(* PLC project Cell Example , CTH FIX1 1.0, author CTH SS2 *)
(* stored: companyURL www.chalmers.se, creationDateTime 2008-03-19T20:31:26, version 1.0, modificationDateTime 2008-09-18T15:59:40, organization SS2, language en-US *)

TYPE BinaryPositions : ();
END_TYPE

TYPE HMIInput : ARRAY[0..0, 1..12] OF BOOL;
END_TYPE

FUNCTION ADD_E : INT
  VAR_INPUT
    Enable : BOOL := FALSE;
    IN1 : INT := 0;
    IN2 : INT := 0;
  END_VAR
  VAR_OUTPUT
    EnableO : BOOL := FALSE;
  END_VAR

(* LD diagram, written out as Structured Text *)
END_FUNCTION

FUNCTION DEC_E : INT
  VAR_INPUT
    Enable : BOOL;
  END_VAR
  VAR_OUTPUT
    EnableO : BOOL;
  END_VAR

(* LD diagram, written out as Structured Text *)
END_FUNCTION

FUNCTION MOVE_E : STRING
  VAR_INPUT
    Enable : BOOL := FALSE;
    IN : STRING;
  END_VAR
  VAR_OUTPUT
    EnableO : BOOL := FALSE;
  END_VAR

(* LD diagram, written out as Structured Text *)
END_FUNCTION

FUNCTION_BLOCK test4
  VAR_INPUT
    i1 : BOOL := FALSE;
  END_VAR
  VAR_OUTPUT
    o1 : BOOL := TRUE;
  END_VAR

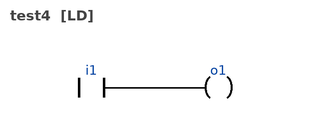
(* LD diagram, written out as Structured Text *)
o1 := i1;
END_FUNCTION_BLOCK

FUNCTION_BLOCK test2
  VAR_INPUT
    i : BOOL;
  END_VAR
  VAR_OUTPUT
    o : BOOL;
  END_VAR
  VAR
    internal1 : test4;
  END_VAR

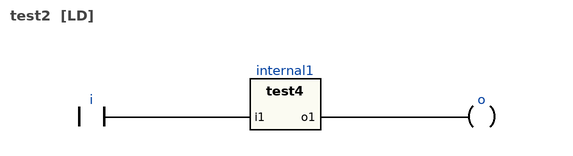
(* LD diagram, written out as Structured Text *)
internal1(i1 := i);
o := internal1.o1;
END_FUNCTION_BLOCK

FUNCTION_BLOCK test5
  VAR_INPUT
    in : BOOL;
  END_VAR
  VAR_OUTPUT
    ut : BOOL;
  END_VAR

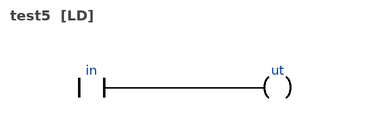
(* LD diagram, written out as Structured Text *)
ut := in;
END_FUNCTION_BLOCK

FUNCTION_BLOCK test3
  VAR_INPUT
    in1 : BOOL;
  END_VAR
  VAR_OUTPUT
    ut1 : BOOL;
  END_VAR
  VAR
    internal1 : test4;
    internal2 : test5;
  END_VAR

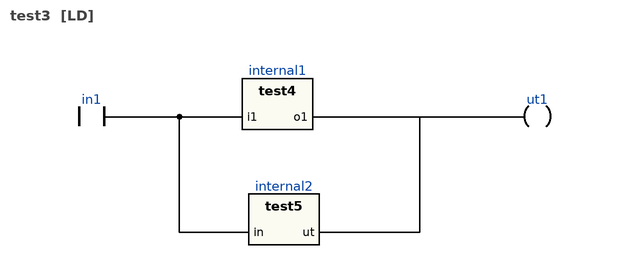
(* LD diagram, written out as Structured Text *)
internal1(i1 := in1);
internal2(in := in1);
ut1 := internal1.o1 OR internal2.ut;
END_FUNCTION_BLOCK

FUNCTION_BLOCK TestFB
  VAR_INPUT
    IN1 : BOOL := FALSE;
    IN2 : INT := 0;
    IN3 : BOOL := FALSE;
  END_VAR
  VAR_OUTPUT
    OUT1 : BOOL := FALSE;
    OUT2 : BOOL := FALSE;
    OUT3 : BOOL := FALSE;
    OUT4 : INT := 0;
  END_VAR
  VAR
    internal1 : test2;
    internal2 : test3;
  END_VAR

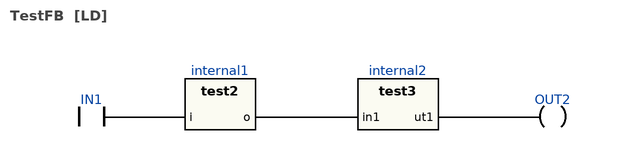
(* LD diagram, written out as Structured Text *)
internal1(i := IN1);
internal2(in1 := internal1.o);
OUT2 := internal2.ut1;
END_FUNCTION_BLOCK

FUNCTION_BLOCK RAC
  VAR_INPUT
    IN1 : BOOL := FALSE;
  END_VAR
  VAR_OUTPUT
    OUT : BOOL := FALSE;
  END_VAR
  VAR_INPUT
    IN2 : BOOL := TRUE;
  END_VAR
  VAR
    Var3 : BOOL := TRUE;
    IN4 : INT := 5;
  END_VAR
  VAR_OUTPUT
    State : STRING := 'Undefined';
  END_VAR
  VAR
    timer : TON;
    passedTime : TIME := 20;
    test : TestFB;
  END_VAR
  VAR_OUTPUT
    OUT2 : BOOL := TRUE;
  END_VAR
  VAR  (* added by the conversion: wires and edge detectors of the diagram *)
    _ADD_E24_ : ANY;
    _ADD_E24_OUT : INT;
    _MOVE_E26_ : ANY;
    _MOVE_E26_OUT : STRING;
    _DEC_E34_ : ANY;
    _DEC_E34_OUT : INT;
  END_VAR

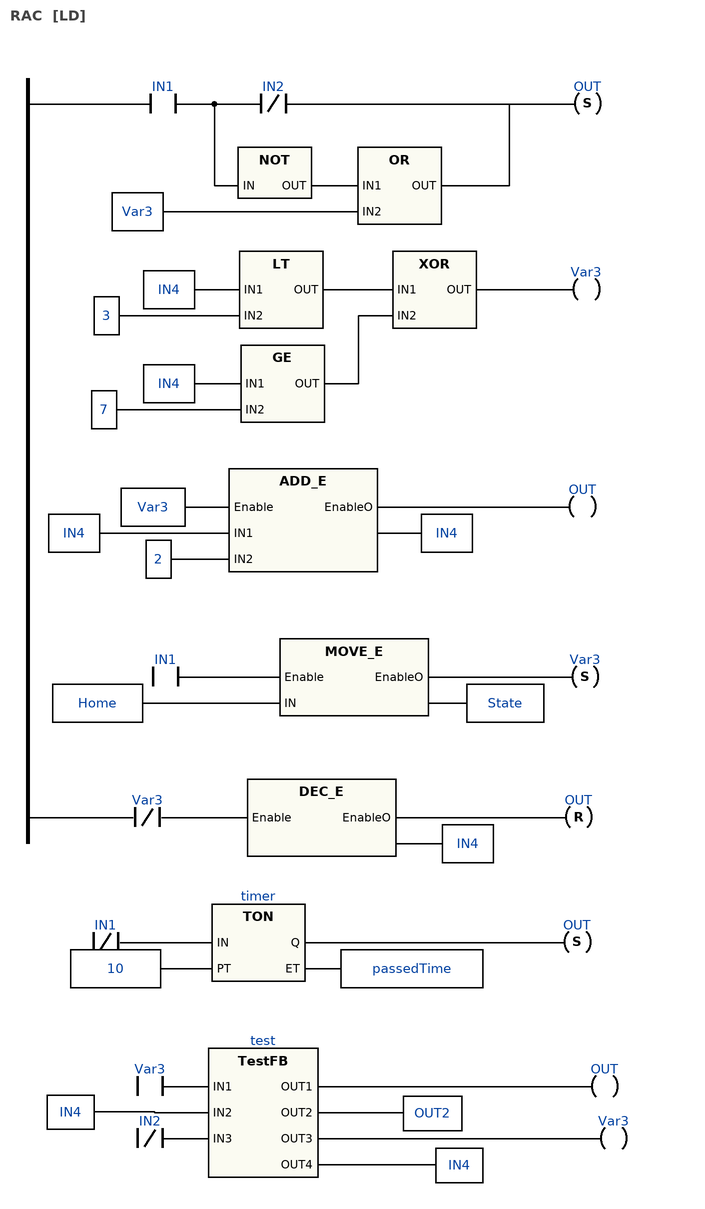
(* LD diagram, written out as Structured Text *)
IF IN1 AND NOT IN2 OR NOT IN1 OR Var3 THEN OUT := TRUE; END_IF;
Var3 := IN4 < 3 XOR IN4 >= 7;
_ADD_E24_OUT := ADD_E(Enable := Var3, IN1 := IN4, IN2 := 2,  => _ADD_E24_);
OUT := _ADD_E24_OUT;
IN4 := _ADD_E24_OUT;
_MOVE_E26_OUT := MOVE_E(Enable := IN1, IN := Home,  => _MOVE_E26_);
IF _MOVE_E26_OUT THEN Var3 := TRUE; END_IF;
State := _MOVE_E26_OUT;
_DEC_E34_OUT := DEC_E(Enable := NOT Var3,  => _DEC_E34_);
IF _DEC_E34_OUT THEN OUT := FALSE; END_IF;
IN4 := _DEC_E34_OUT;
timer(IN := NOT IN1, PT := 10);
IF timer.Q THEN OUT := TRUE; END_IF;
passedTime := timer.ET;
test(IN1 := Var3, IN2 := IN4, IN3 := NOT IN2);
OUT := test.OUT1;
OUT2 := test.OUT2;
Var3 := test.OUT3;
IN4 := test.OUT4;
END_FUNCTION_BLOCK

FUNCTION MOV_M : INT
  VAR_INPUT
    Enable : BOOL := FALSE;
    s_in : INT := 0;
  END_VAR
  VAR_OUTPUT
    EnableO : BOOL := FALSE;
  END_VAR

(* LD diagram, written out as Structured Text *)
END_FUNCTION

FUNCTION INCP_M : INT
  VAR_INPUT
    Enable : BOOL := FALSE;
  END_VAR
  VAR_OUTPUT
    EnableO : BOOL := FALSE;
  END_VAR

(* LD diagram, written out as Structured Text *)
END_FUNCTION

FUNCTION_BLOCK ESTOP
  VAR_INPUT
    ResetType : BOOL := FALSE;
    ChannelA : BOOL := TRUE;
    ChannelB : BOOL := TRUE;
    CircuitReset : BOOL := FALSE;
    FaultReset : BOOL := FALSE;
  END_VAR
  VAR_OUTPUT
    O1 : BOOL := FALSE;
    CI : BOOL := FALSE;
    CRHO : BOOL := FALSE;
    II : BOOL := FALSE;
    FP : BOOL := FALSE;
  END_VAR
  VAR
    RstOnlyByA : BOOL := FALSE;
    RstOnlyByB : BOOL := FALSE;
    RisingEdge1 : R_TRIG;
    RisingEdge2 : R_TRIG;
    Timer2 : TON;
    Timer1 : TON;
    RisingEdge3 : R_TRIG;
  END_VAR

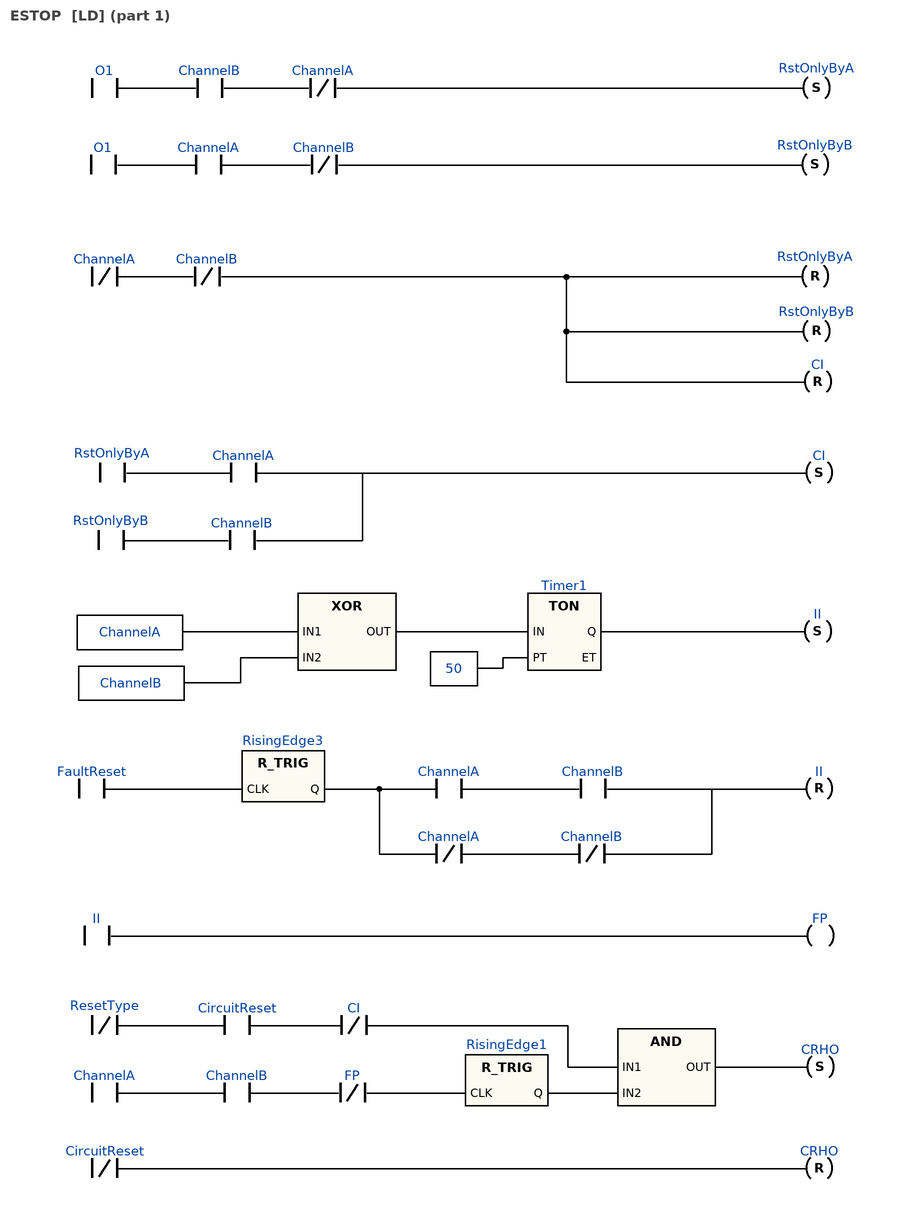
(* LD diagram, written out as Structured Text *)
IF O1 AND ChannelB AND NOT ChannelA THEN RstOnlyByA := TRUE; END_IF;
IF O1 AND ChannelA AND NOT ChannelB THEN RstOnlyByB := TRUE; END_IF;
IF NOT ChannelA AND NOT ChannelB THEN RstOnlyByA := FALSE; END_IF;
IF NOT ChannelA AND NOT ChannelB THEN RstOnlyByB := FALSE; END_IF;
IF NOT ChannelA AND NOT ChannelB THEN CI := FALSE; END_IF;
IF RstOnlyByA AND ChannelA OR RstOnlyByB AND ChannelB THEN CI := TRUE; END_IF;
Timer1(IN := ChannelA XOR ChannelB, PT := 50);
IF Timer1.Q THEN II := TRUE; END_IF;
RisingEdge3(CLK := FaultReset);
IF RisingEdge3.Q AND (ChannelA AND ChannelB OR NOT ChannelA AND NOT ChannelB) THEN II := FALSE; END_IF;
FP := II;
RisingEdge1(CLK := ChannelA AND ChannelB AND NOT FP);
IF NOT ResetType AND CircuitReset AND NOT CI AND RisingEdge1.Q THEN CRHO := TRUE; END_IF;
IF NOT CircuitReset THEN CRHO := FALSE; END_IF;
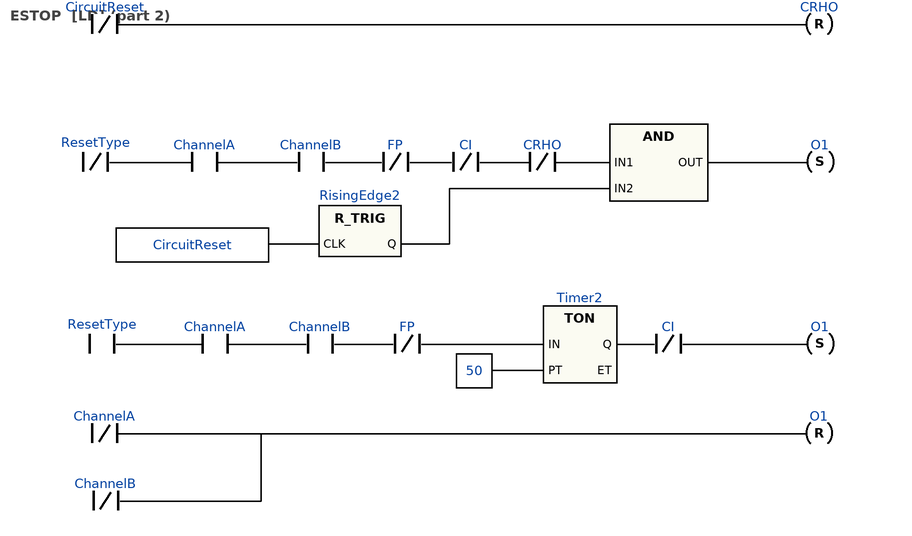
RisingEdge2(CLK := CircuitReset);
IF NOT ResetType AND ChannelA AND ChannelB AND NOT FP AND NOT CI AND NOT CRHO AND RisingEdge2.Q THEN O1 := TRUE; END_IF;
Timer2(IN := ResetType AND ChannelA AND ChannelB AND NOT FP, PT := 50);
IF Timer2.Q AND NOT CI THEN O1 := TRUE; END_IF;
IF NOT ChannelA OR NOT ChannelB THEN O1 := FALSE; END_IF;
END_FUNCTION_BLOCK

FUNCTION_BLOCK ENPEN
  VAR_INPUT
    ResetType : BOOL := FALSE;
    ChannelA : BOOL := TRUE;
    ChannelB : BOOL := TRUE;
    CircuitReset : BOOL := FALSE;
    FaultReset : BOOL := FALSE;
  END_VAR
  VAR_OUTPUT
    O1 : BOOL := FALSE;
    CI : BOOL := FALSE;
    CRHO : BOOL := FALSE;
    II : BOOL := FALSE;
    FP : BOOL := FALSE;
  END_VAR
  VAR
    RstOnlyByA : BOOL := FALSE;
    RstOnlyByB : BOOL := FALSE;
    CircuitReset_pre : BOOL := FALSE;
    RisingEdge1 : R_TRIG;
    RisingEdge2 : R_TRIG;
    Timer2 : TON;
    Timer1 : TON;
  END_VAR

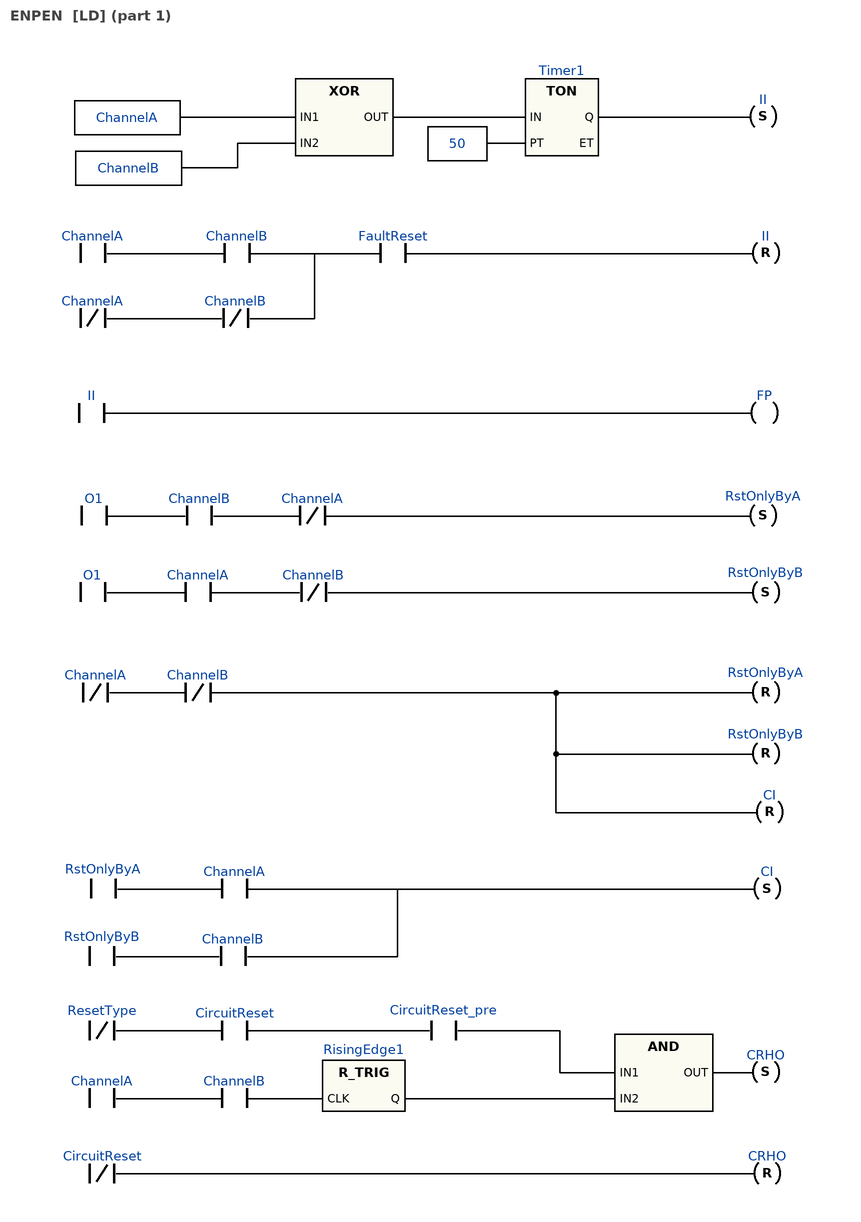
(* LD diagram, written out as Structured Text *)
Timer1(IN := ChannelA XOR ChannelB, PT := 50);
IF Timer1.Q THEN II := TRUE; END_IF;
IF (ChannelA AND ChannelB OR NOT ChannelA AND NOT ChannelB) AND FaultReset THEN II := FALSE; END_IF;
FP := II;
IF O1 AND ChannelB AND NOT ChannelA THEN RstOnlyByA := TRUE; END_IF;
IF O1 AND ChannelA AND NOT ChannelB THEN RstOnlyByB := TRUE; END_IF;
IF NOT ChannelA AND NOT ChannelB THEN RstOnlyByA := FALSE; END_IF;
IF NOT ChannelA AND NOT ChannelB THEN RstOnlyByB := FALSE; END_IF;
IF NOT ChannelA AND NOT ChannelB THEN CI := FALSE; END_IF;
IF RstOnlyByA AND ChannelA OR RstOnlyByB AND ChannelB THEN CI := TRUE; END_IF;
RisingEdge1(CLK := ChannelA AND ChannelB);
IF NOT ResetType AND CircuitReset AND CircuitReset_pre AND RisingEdge1.Q THEN CRHO := TRUE; END_IF;
IF NOT CircuitReset THEN CRHO := FALSE; END_IF;
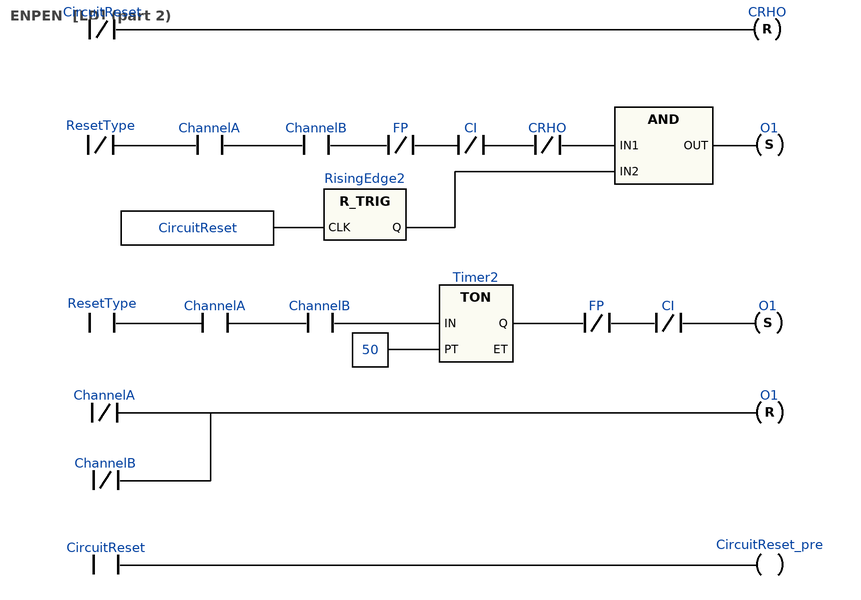
RisingEdge2(CLK := CircuitReset);
IF NOT ResetType AND ChannelA AND ChannelB AND NOT FP AND NOT CI AND NOT CRHO AND RisingEdge2.Q THEN O1 := TRUE; END_IF;
Timer2(IN := ResetType AND ChannelA AND ChannelB, PT := 50);
IF Timer2.Q AND NOT FP AND NOT CI THEN O1 := TRUE; END_IF;
IF NOT ChannelA OR NOT ChannelB THEN O1 := FALSE; END_IF;
CircuitReset_pre := CircuitReset;
END_FUNCTION_BLOCK

FUNCTION_BLOCK FPMS
  VAR
    NMCondition : BOOL := FALSE;
    MMSCondition : BOOL := FALSE;
  END_VAR
  VAR_INPUT
    FaultReset : BOOL := FALSE;
  END_VAR
  VAR_OUTPUT
    NM : BOOL := FALSE;
    FP : BOOL := FALSE;
  END_VAR
  VAR
    Timer1 : TON;
  END_VAR
  VAR_INPUT
    Input1 : BOOL := FALSE;
    Input2 : BOOL := FALSE;
    Input3 : BOOL := FALSE;
    Input4 : BOOL := FALSE;
    Input5 : BOOL := FALSE;
  END_VAR
  VAR_OUTPUT
    MMS : BOOL := FALSE;
  END_VAR
  VAR
    Timer2 : TON;
  END_VAR
  VAR_OUTPUT
    O1 : BOOL := FALSE;
    O2 : BOOL := FALSE;
    O3 : BOOL := FALSE;
    O4 : BOOL := FALSE;
    O5 : BOOL := FALSE;
  END_VAR
  VAR
    RisingEdge1 : R_TRIG;
    RisingEdge2 : R_TRIG;
  END_VAR

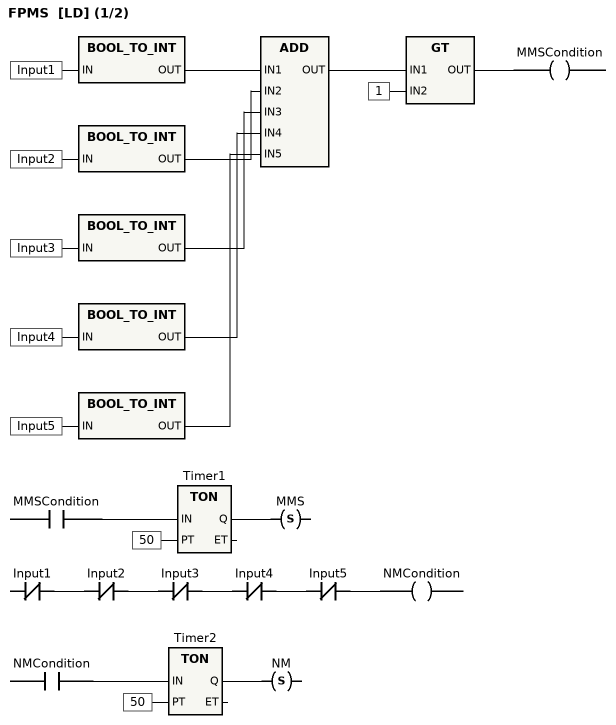
(* LD diagram, written out as Structured Text *)
MMSCondition := BOOL_TO_INT(Input1) + BOOL_TO_INT(Input2) + BOOL_TO_INT(Input3) + BOOL_TO_INT(Input4) + BOOL_TO_INT(Input5) > 1;
NMCondition := NOT Input1 AND NOT Input2 AND NOT Input3 AND NOT Input4 AND NOT Input5;
Timer1(IN := MMSCondition, PT := 50);
IF Timer1.Q THEN MMS := TRUE; END_IF;
Timer2(IN := NMCondition, PT := 50);
IF Timer2.Q THEN NM := TRUE; END_IF;
RisingEdge1(CLK := FaultReset);
IF RisingEdge1.Q AND NOT NMCondition THEN NM := FALSE; END_IF;
RisingEdge2(CLK := FaultReset);
IF RisingEdge2.Q AND NOT MMSCondition THEN MMS := FALSE; END_IF;
FP := NM OR MMS;
O1 := Input1 AND NOT Input2 AND NOT Input3 AND NOT Input4 AND NOT Input5 OR (NMCondition OR MMSCondition) AND O1;
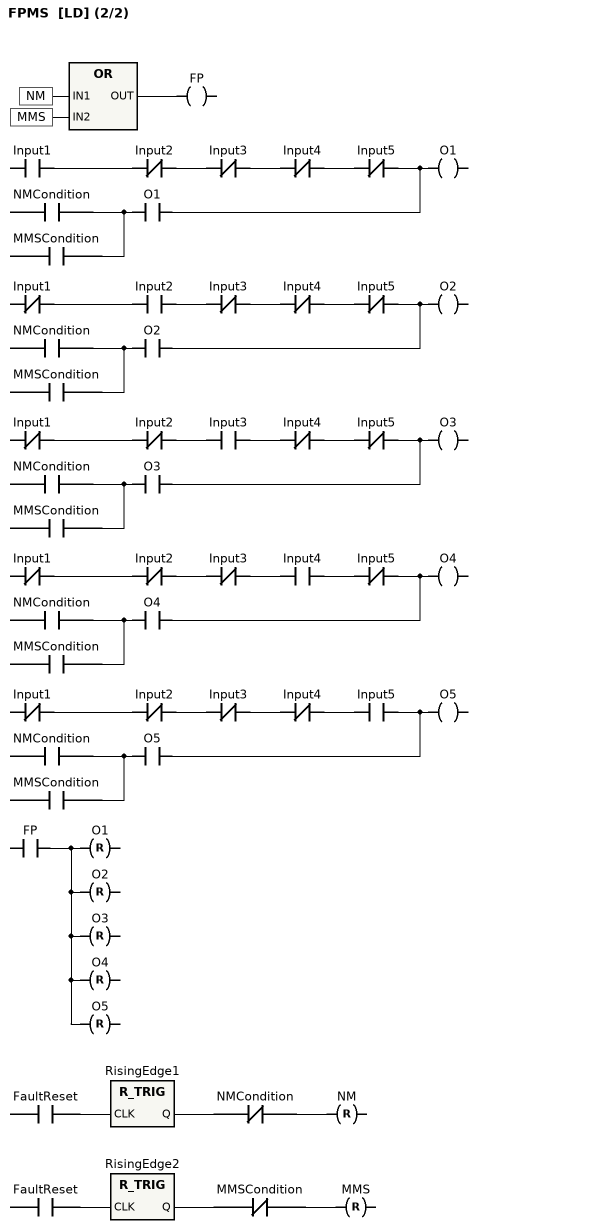
O2 := NOT Input1 AND Input2 AND NOT Input3 AND NOT Input4 AND NOT Input5 OR (NMCondition OR MMSCondition) AND O2;
O3 := NOT Input1 AND NOT Input2 AND Input3 AND NOT Input4 AND NOT Input5 OR (NMCondition OR MMSCondition) AND O3;
O4 := NOT Input1 AND NOT Input2 AND NOT Input3 AND Input4 AND NOT Input5 OR (NMCondition OR MMSCondition) AND O4;
O5 := NOT Input1 AND NOT Input2 AND NOT Input3 AND NOT Input4 AND Input5 OR (NMCondition OR MMSCondition) AND O5;
IF FP THEN O1 := FALSE; END_IF;
IF FP THEN O2 := FALSE; END_IF;
IF FP THEN O3 := FALSE; END_IF;
IF FP THEN O4 := FALSE; END_IF;
IF FP THEN O5 := FALSE; END_IF;
END_FUNCTION_BLOCK

FUNCTION_BLOCK RIN
  VAR_INPUT
    ResetType : BOOL := FALSE;
    ChannelA : BOOL := TRUE;
    ChannelB : BOOL := TRUE;
    CircuitReset : BOOL := FALSE;
    FaultReset : BOOL := FALSE;
  END_VAR
  VAR_OUTPUT
    O1 : BOOL := FALSE;
    CI : BOOL := FALSE;
    CRHO : BOOL := FALSE;
    II : BOOL := FALSE;
    FP : BOOL := FALSE;
  END_VAR
  VAR
    RstOnlyByA : BOOL := FALSE;
    RstOnlyByB : BOOL := FALSE;
    CircuitReset_pre : BOOL := FALSE;
    RisingEdge1 : R_TRIG;
    RisingEdge2 : R_TRIG;
    Timer2 : TON;
    Timer1 : TON;
  END_VAR
  VAR_TEMP
    Spec_SettingO1 : BOOL;
    Spec_ResettingO1 : BOOL;
    Spec_NotSettingO1 : BOOL;
    O1_previous : BOOL;
  END_VAR

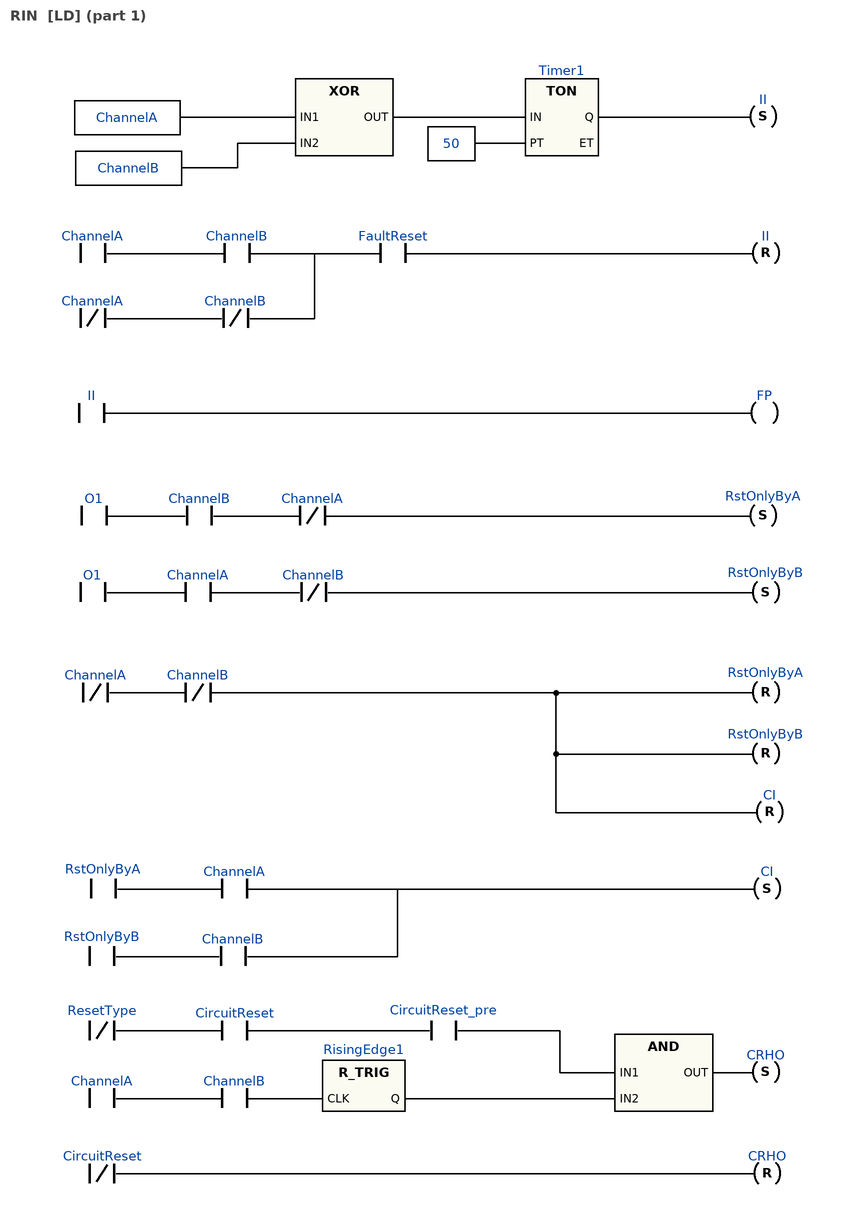
(* LD diagram, written out as Structured Text *)
Timer1(IN := ChannelA XOR ChannelB, PT := 50);
IF Timer1.Q THEN II := TRUE; END_IF;
IF (ChannelA AND ChannelB OR NOT ChannelA AND NOT ChannelB) AND FaultReset THEN II := FALSE; END_IF;
FP := II;
IF O1 AND ChannelB AND NOT ChannelA THEN RstOnlyByA := TRUE; END_IF;
IF O1 AND ChannelA AND NOT ChannelB THEN RstOnlyByB := TRUE; END_IF;
IF NOT ChannelA AND NOT ChannelB THEN RstOnlyByA := FALSE; END_IF;
IF NOT ChannelA AND NOT ChannelB THEN RstOnlyByB := FALSE; END_IF;
IF NOT ChannelA AND NOT ChannelB THEN CI := FALSE; END_IF;
IF RstOnlyByA AND ChannelA OR RstOnlyByB AND ChannelB THEN CI := TRUE; END_IF;
RisingEdge1(CLK := ChannelA AND ChannelB);
IF NOT ResetType AND CircuitReset AND CircuitReset_pre AND RisingEdge1.Q THEN CRHO := TRUE; END_IF;
IF NOT CircuitReset THEN CRHO := FALSE; END_IF;
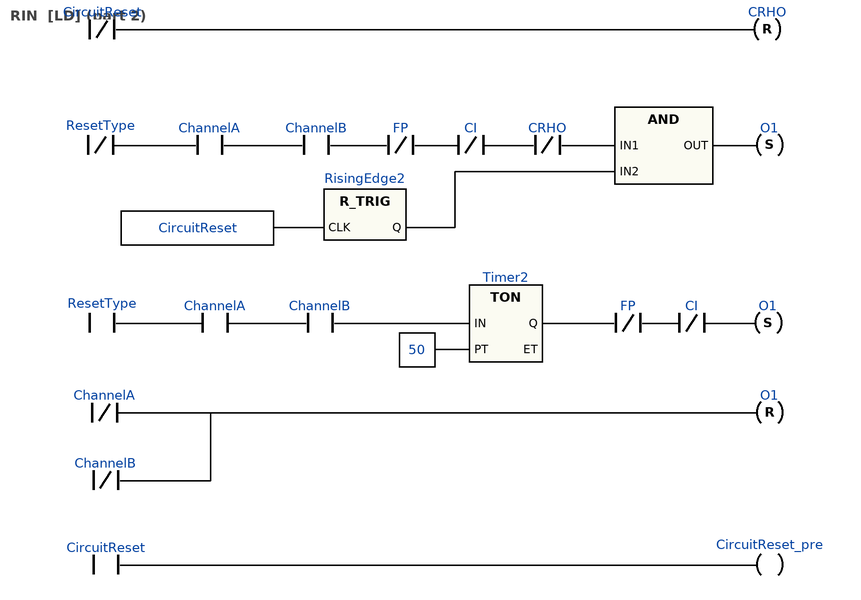
RisingEdge2(CLK := CircuitReset);
IF NOT ResetType AND ChannelA AND ChannelB AND NOT FP AND NOT CI AND NOT CRHO AND RisingEdge2.Q THEN O1 := TRUE; END_IF;
Timer2(IN := ResetType AND ChannelA AND ChannelB, PT := 50);
IF Timer2.Q AND NOT FP AND NOT CI THEN O1 := TRUE; END_IF;
IF NOT ChannelA OR NOT ChannelB THEN O1 := FALSE; END_IF;
CircuitReset_pre := CircuitReset;
END_FUNCTION_BLOCK

FUNCTION Always : BOOL
  VAR_INPUT
     : BOOL;
  END_VAR

(* LD diagram, written out as Structured Text *)
END_FUNCTION

FUNCTION Sometime : BOOL
  VAR_INPUT
     : BOOL;
  END_VAR

(* LD diagram, written out as Structured Text *)
END_FUNCTION

FUNCTION Never : BOOL
  VAR_INPUT
     : BOOL;
  END_VAR

(* LD diagram, written out as Structured Text *)
END_FUNCTION

FUNCTION Imply : BOOL
  VAR_INPUT
    IfTrue : BOOL;
    ThenTrue : BOOL;
  END_VAR

(* LD diagram, written out as Structured Text *)
END_FUNCTION

FUNCTION SteadyExpressionT : BOOL
  VAR_INPUT
    HeldTrueForXMilliSeconds : BOOL;
    X : INT := 10;
  END_VAR

(* LD diagram, written out as Structured Text *)
END_FUNCTION

FUNCTION SteadyExpressionSC : BOOL
  VAR_INPUT
    RemainTrueForXScanCycles : BOOL;
    X : INT := 1;
  END_VAR

(* LD diagram, written out as Structured Text *)
END_FUNCTION

FUNCTION_BLOCK Implies
  VAR_INPUT
    IfTrue : BOOL;
  END_VAR
  VAR_OUTPUT
    ThenTrue : BOOL;
  END_VAR

(* LD diagram, written out as Structured Text *)
END_FUNCTION_BLOCK

FUNCTION WhileNot : BOOL
  VAR_INPUT
    RemainTrue : BOOL;
    WhileNot : BOOL;
  END_VAR

(* LD diagram, written out as Structured Text *)
END_FUNCTION

FUNCTION MOV_E_Int : INT
  VAR_INPUT
    Enable : BOOL := FALSE;
    Source : INT := 0;
  END_VAR
  VAR_OUTPUT
    EnableO : BOOL := FALSE;
  END_VAR

(* LD diagram, written out as Structured Text *)
END_FUNCTION

FUNCTION_BLOCK TOF_RSLogix
  VAR_INPUT
    TimerOffDelay : BOOL;
    Preset : INT;
  END_VAR
  VAR_OUTPUT
    EnableO : BOOL := FALSE;
    DN : BOOL := FALSE;
    ACC : INT := 0;
    TT : BOOL := FALSE;
  END_VAR
  VAR
    TON1 : TON;
  END_VAR

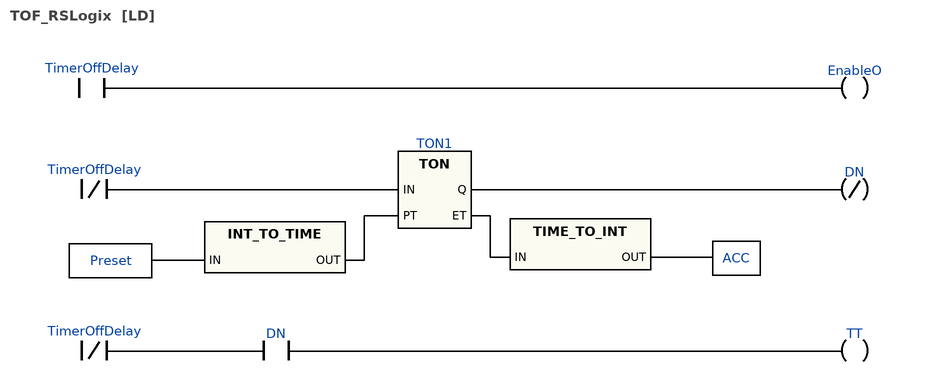
(* LD diagram, written out as Structured Text *)
EnableO := TimerOffDelay;
TON1(IN := NOT TimerOffDelay, PT := INT_TO_TIME(Preset));
DN := NOT TON1.Q;
ACC := TIME_TO_INT(TON1.ET);
TT := NOT TimerOffDelay AND DN;
END_FUNCTION_BLOCK

FUNCTION_BLOCK TON_RSLogix
  VAR_INPUT
    TimerOnDelay : BOOL := FALSE;
    Preset : INT := 0;
  END_VAR
  VAR_OUTPUT
    EnableO : BOOL := FALSE;
    DN : BOOL := FALSE;
    ACC : INT := 0;
    TT : BOOL := FALSE;
  END_VAR
  VAR
    TON1 : TON;
  END_VAR

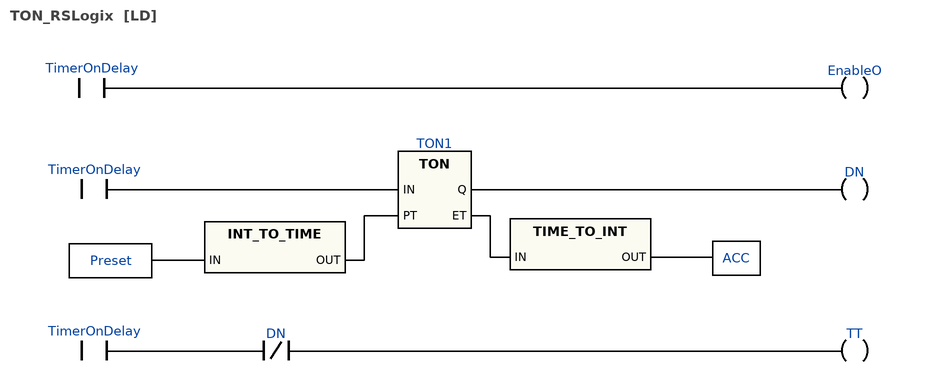
(* LD diagram, written out as Structured Text *)
EnableO := TimerOnDelay;
TON1(IN := TimerOnDelay, PT := INT_TO_TIME(Preset));
DN := TON1.Q;
ACC := TIME_TO_INT(TON1.ET);
TT := TimerOnDelay AND NOT DN;
END_FUNCTION_BLOCK

FUNCTION_BLOCK HMI_Safety
  VAR_IN_OUT
    ESTOP_FP : BOOL := FALSE;
    CommOK : BOOL := FALSE;
  END_VAR
  VAR_INPUT
    FirstScanOneShot : BOOL;
    NoEStopCHA : BOOL;
    NoEStopCHB : BOOL;
  END_VAR
  VAR_OUTPUT
    ESTOP_FaultReset : BOOL := FALSE;
    ESTOP_O1 : BOOL := FALSE;
    NoEstop : BOOL := FALSE;
  END_VAR
  VAR_INPUT
    AutoModeS : BOOL;
    ManModeS : BOOL;
  END_VAR
  VAR_IN_OUT
    AutoMan_FP : BOOL := FALSE;
  END_VAR
  VAR_OUTPUT
    AutoMan_FaultReset : BOOL := FALSE;
    AutoManDebounce_PRE : INT := 200;
    AutoManDebounce_TT : BOOL := FALSE;
  END_VAR
  VAR_IN_OUT
    Pos1Int : BOOL := FALSE;
    Pos2Int : BOOL := FALSE;
  END_VAR
  VAR_OUTPUT
    AutoMan_O1 : BOOL := FALSE;
    AutoMan_O2 : BOOL := FALSE;
    AutoMode : BOOL := FALSE;
    ManualMode : BOOL := FALSE;
  END_VAR
  VAR_IN_OUT
    PendantOK_FP : BOOL := FALSE;
  END_VAR
  VAR_OUTPUT
    PendantOK_FaultReset : BOOL := FALSE;
  END_VAR
  VAR_INPUT
    E130CREP : BOOL;
    E134CREP : BOOL;
    HMI_Select : BOOL;
  END_VAR
  VAR_IN_OUT
    Selected : BOOL := FALSE;
  END_VAR
  VAR_INPUT
    HMI_SelectionOK : BOOL;
    Gates_SelectAvail : BOOL;
    EnablePB : BOOL;
  END_VAR
  VAR_IN_OUT
    Enable : BOOL := FALSE;
    PHMIEnable : BOOL := FALSE;
    EnableAntiRepeat : BOOL := FALSE;
  END_VAR
  VAR_OUTPUT
    EnableTmr_PRE : INT := 600;
    EnableTmr_DN : BOOL := FALSE;
  END_VAR
  VAR_INPUT
    OneHMIEnabled : BOOL;
    Gates_OneRobotToolMinorReq : BOOL;
    OneHMIMode : BOOL;
  END_VAR
  VAR_OUTPUT
    PendEnable : BOOL := FALSE;
    PendOk : BOOL := FALSE;
  END_VAR
  VAR_INPUT
    AlwaysOff : BOOL;
    FltBcn : BOOL;
  END_VAR
  VAR_OUTPUT
    O_FaultLT : BOOL := FALSE;
  END_VAR
  VAR_INPUT
    ResetLT : BOOL;
  END_VAR
  VAR_OUTPUT
    O_ResetLT : BOOL := FALSE;
  END_VAR
  VAR_INPUT
    AutoInitLT : BOOL;
  END_VAR
  VAR_OUTPUT
    O_AutoInitLT : BOOL := FALSE;
  END_VAR
  VAR_INPUT
    CombinedStatus : BOOL;
  END_VAR
  VAR_OUTPUT
    NoSafetyFaults : BOOL := FALSE;
  END_VAR
  VAR_IN_OUT
    BackCheck_NoEStop : BOOL := FALSE;
    BackCheck_NoSafetyFaults : BOOL := FALSE;
  END_VAR
  VAR
    ESTOP1 : ESTOP;
    TOF1 : TOF_RSLogix;
    FPMS1 : FPMS;
    ENPEN1 : ENPEN;
    TON1 : TON_RSLogix;
  END_VAR
  VAR_OUTPUT
    ESTOP_CI : BOOL := FALSE;
    ESTOP_CRHO : BOOL := FALSE;
    ESTOP_II : BOOL := FALSE;
  END_VAR
  VAR  (* added by the conversion: wires and edge detectors of the diagram *)
    _MOV_E_Int30_ : ANY;
    _MOV_E_Int30_OUT : INT;
    _MOV_E_Int83_ : ANY;
    _MOV_E_Int83_OUT : INT;
  END_VAR

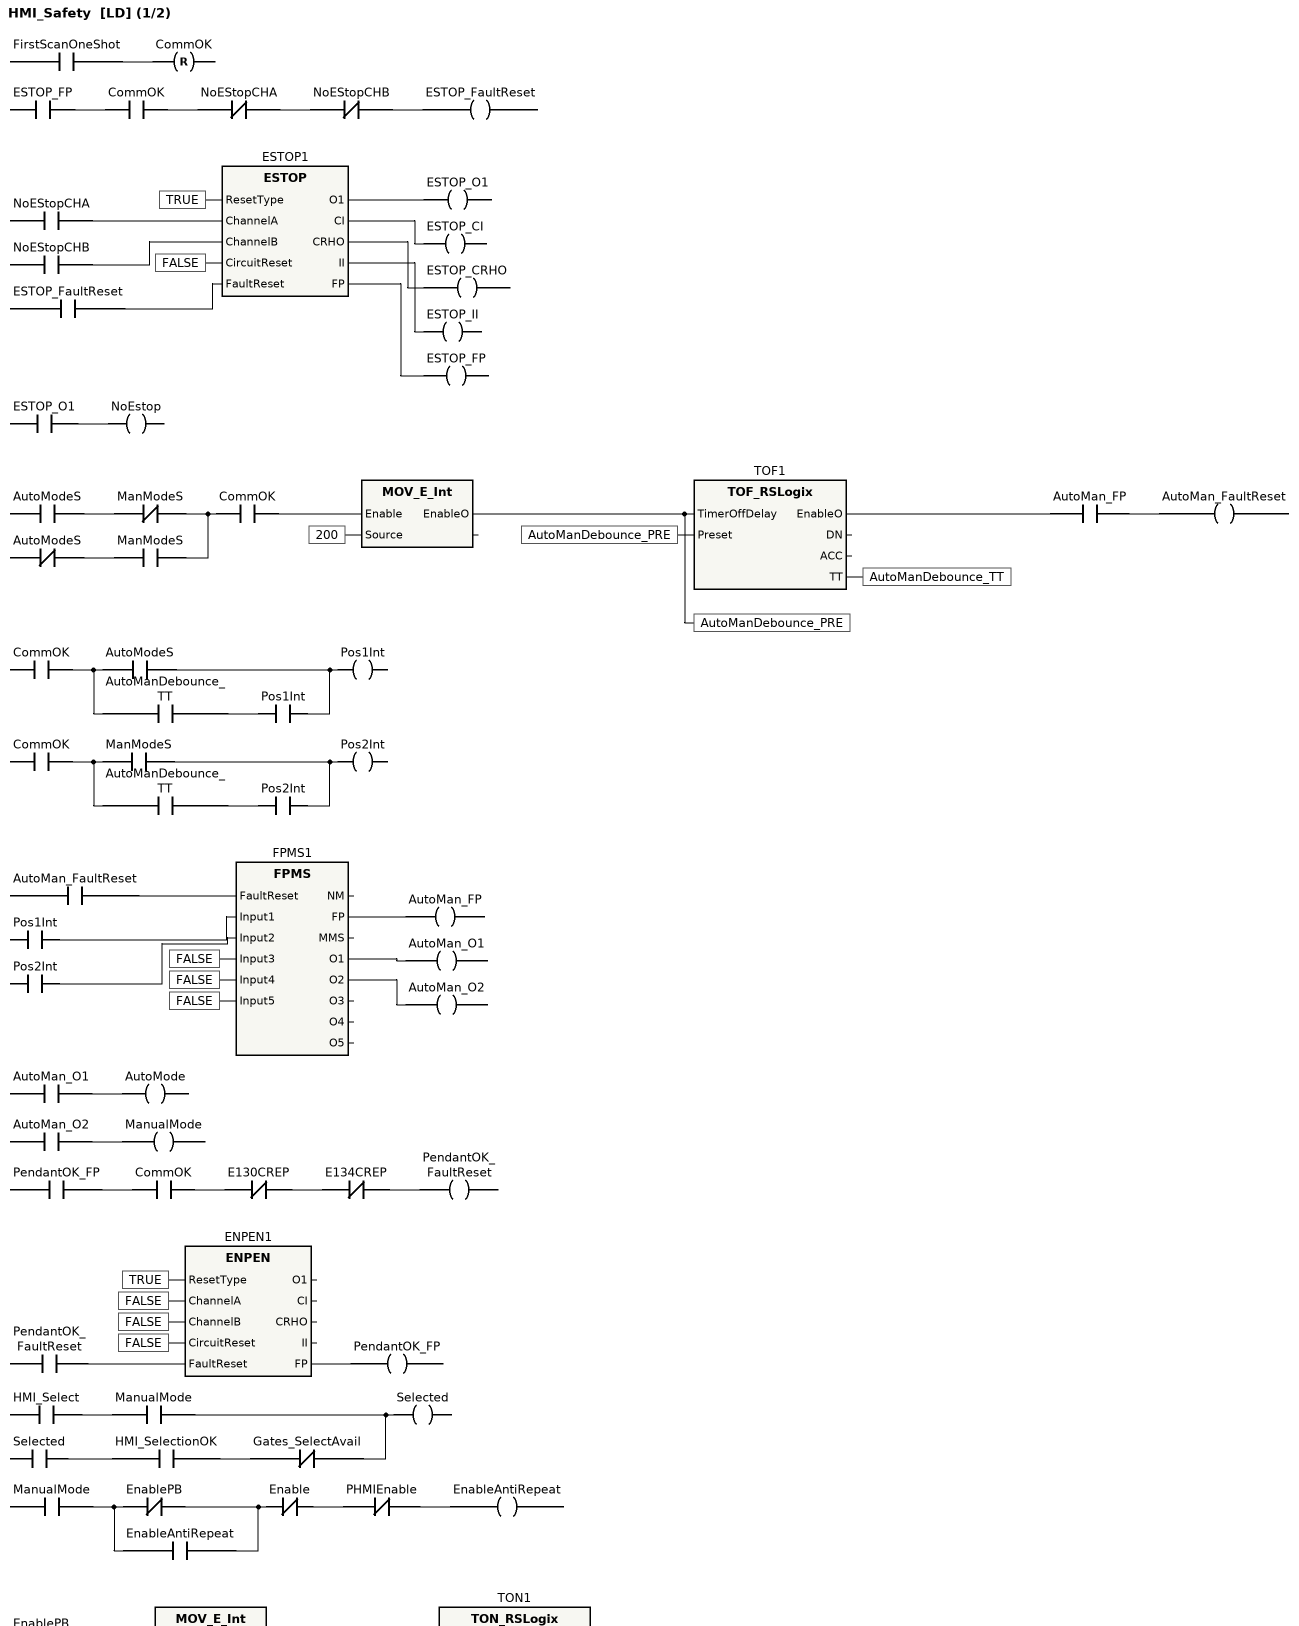
(* LD diagram, written out as Structured Text *)
IF FirstScanOneShot THEN CommOK := FALSE; END_IF;
ESTOP_FaultReset := ESTOP_FP AND CommOK AND NOT NoEStopCHA AND NOT NoEStopCHB;
ESTOP1(ResetType := TRUE, ChannelA := NoEStopCHA, ChannelB := NoEStopCHB, CircuitReset := FALSE, FaultReset := ESTOP_FaultReset);
ESTOP_O1 := ESTOP1.O1;
ESTOP_CI := ESTOP1.CI;
ESTOP_CRHO := ESTOP1.CRHO;
ESTOP_II := ESTOP1.II;
ESTOP_FP := ESTOP1.FP;
NoEstop := ESTOP_O1;
_MOV_E_Int30_OUT := MOV_E_Int(Enable := (AutoModeS AND NOT ManModeS OR NOT AutoModeS AND ManModeS) AND CommOK, Source := 200,  => _MOV_E_Int30_);
TOF1(TimerOffDelay := _MOV_E_Int30_OUT, Preset := AutoManDebounce_PRE);
AutoMan_FaultReset := TOF1.EnableO AND AutoMan_FP;
AutoManDebounce_PRE := _MOV_E_Int30_OUT;
AutoManDebounce_TT := TOF1.TT;
Pos1Int := CommOK AND (AutoModeS OR AutoManDebounce_TT AND Pos1Int);
Pos2Int := CommOK AND (ManModeS OR AutoManDebounce_TT AND Pos2Int);
FPMS1(FaultReset := AutoMan_FaultReset, Input1 := Pos1Int, Input2 := Pos2Int, Input3 := FALSE, Input4 := FALSE, Input5 := FALSE);
AutoMan_FP := FPMS1.FP;
AutoMan_O1 := FPMS1.O1;
AutoMan_O2 := FPMS1.O2;
AutoMode := AutoMan_O1;
ManualMode := AutoMan_O2;
PendantOK_FaultReset := PendantOK_FP AND CommOK AND NOT E130CREP AND NOT E134CREP;
ENPEN1(ResetType := TRUE, ChannelA := FALSE, ChannelB := FALSE, CircuitReset := FALSE, FaultReset := PendantOK_FaultReset);
PendantOK_FP := ENPEN1.FP;
Selected := HMI_Select AND ManualMode OR Selected AND HMI_SelectionOK AND NOT Gates_SelectAvail;
EnableAntiRepeat := ManualMode AND (NOT EnablePB OR EnableAntiRepeat) AND NOT Enable AND NOT PHMIEnable;
_MOV_E_Int83_OUT := MOV_E_Int(Enable := EnablePB, Source := 600,  => _MOV_E_Int83_);
EnableTmr_PRE := _MOV_E_Int83_OUT;
TON1(TimerOnDelay := _MOV_E_Int83_OUT, Preset := EnableTmr_PRE);
EnableTmr_DN := TON1.DN;
Enable := ManualMode AND NOT EnableTmr_DN AND (EnableAntiRepeat OR Enable) AND EnablePB AND ((NOT Gates_OneRobotToolMinorReq OR Selected AND HMI_SelectionOK) AND OneHMIEnabled OR (Selected AND HMI_SelectionOK OR NOT Gates_OneRobotToolMinorReq) AND NOT OneHMIMode);
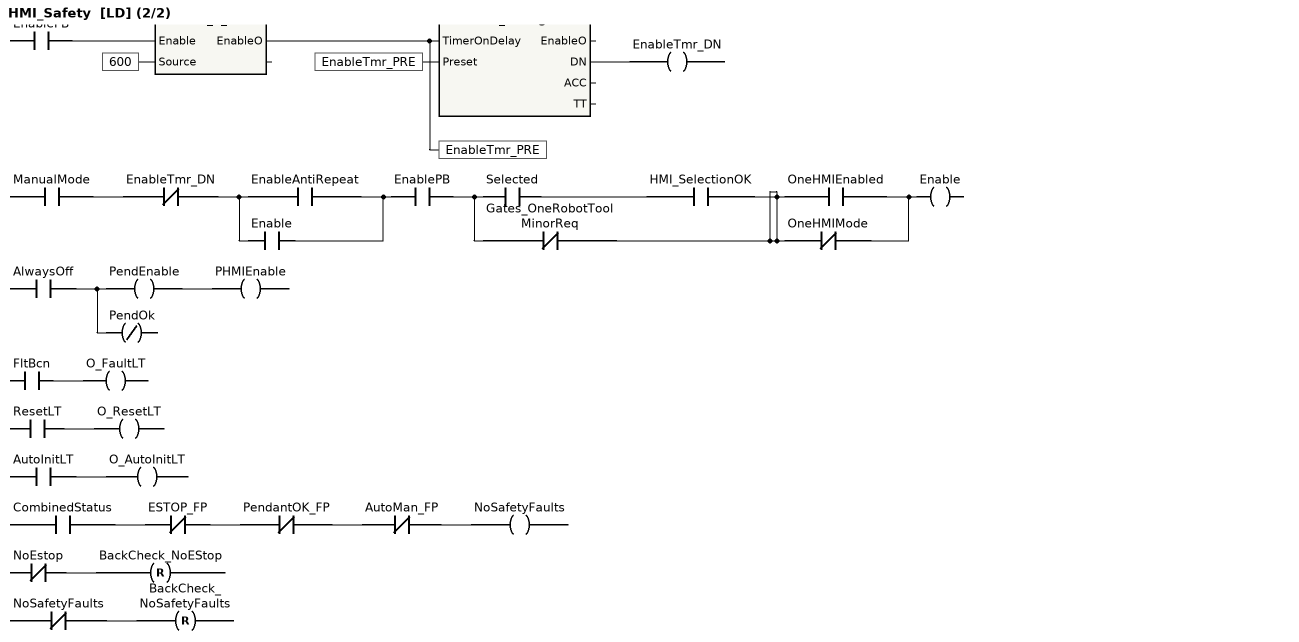
PendEnable := AlwaysOff;
PHMIEnable := AlwaysOff;
PendOk := NOT AlwaysOff;
O_FaultLT := FltBcn;
O_ResetLT := ResetLT;
O_AutoInitLT := AutoInitLT;
NoSafetyFaults := CombinedStatus AND NOT ESTOP_FP AND NOT PendantOK_FP AND NOT AutoMan_FP;
IF NOT NoEstop THEN BackCheck_NoEStop := FALSE; END_IF;
IF NOT NoSafetyFaults THEN BackCheck_NoSafetyFaults := FALSE; END_IF;
END_FUNCTION_BLOCK

FUNCTION_BLOCK PermGuard_Safety
  VAR_IN_OUT
    MuteSw12_FP : BOOL := FALSE;
    CommOK : BOOL := FALSE;
  END_VAR
  VAR_INPUT
    FirstScanOneShot : BOOL;
    SD1ClearChA : BOOL;
    SD1ClearChB : BOOL;
  END_VAR
  VAR_OUTPUT
    MuteSw12_FaultReset : BOOL := FALSE;
    MuteSw12_O1 : BOOL := FALSE;
  END_VAR
  VAR_INPUT
    AutoModeSS : BOOL;
    OverrideModeSS : BOOL;
  END_VAR
  VAR_IN_OUT
    AutoOverride_FP : BOOL := FALSE;
  END_VAR
  VAR_OUTPUT
    AutoOverride_FaultReset : BOOL := FALSE;
    AutoOverrideDebounce_PRE : INT := 50;
    AutoOverrideDebounce_TT : BOOL := FALSE;
  END_VAR
  VAR_IN_OUT
    Pos1Int : BOOL := FALSE;
    Pos2Int : BOOL := FALSE;
  END_VAR
  VAR_OUTPUT
    AutoOverride_O1 : BOOL := FALSE;
    AutoOverride_O2 : BOOL := FALSE;
  END_VAR
  VAR_IN_OUT
    GuardRst_FP : BOOL := FALSE;
  END_VAR
  VAR_OUTPUT
    GuardRst_FaultReset : BOOL := FALSE;
    OverrideLimit_PRE : INT := 50;
    OverrideLimit_DN : BOOL := FALSE;
  END_VAR
  VAR_INPUT
    CombinedStatus : BOOL;
  END_VAR
  VAR_OUTPUT
    NoSafetyFaults : BOOL := FALSE;
  END_VAR
  VAR_IN_OUT
    BackCheck_OneRobotEnable : BOOL := FALSE;
    BackCheck_NoSafetyFaults : BOOL := FALSE;
  END_VAR
  VAR
    MuteSw12 : ENPEN;
    AutoOverrideDebounce : TOF_RSLogix;
    AutoOverride : FPMS;
    GuardRst : RIN;
    OverrideLimit : TON_RSLogix;
  END_VAR
  VAR_OUTPUT
    MuteSw12_CI : BOOL := FALSE;
    MuteSw12_CRHO : BOOL := FALSE;
    MuteSw12_II : BOOL := FALSE;
  END_VAR
  VAR_INPUT
    P1 : BOOL;
    P2 : BOOL;
    P3 : BOOL;
    P4 : BOOL;
  END_VAR
  VAR_IN_OUT
    MuteSw34_FP : BOOL := FALSE;
  END_VAR
  VAR_OUTPUT
    MuteSw34_FaultReset : BOOL := FALSE;
    MuteSw34_O1 : BOOL := FALSE;
    MuteSw34_CI : BOOL := FALSE;
    MuteSw34_CRHO : BOOL := FALSE;
    MuteSw34_II : BOOL := FALSE;
  END_VAR
  VAR
    MuteSw34 : ENPEN;
  END_VAR
  VAR_INPUT
    MutingStatus : BOOL;
  END_VAR
  VAR_OUTPUT
    MuteSD : BOOL := FALSE;
    SDMuteLt : BOOL := FALSE;
  END_VAR
  VAR_INPUT
    LampTest : BOOL;
  END_VAR
  VAR_IN_OUT
    SD1_FP : BOOL := FALSE;
  END_VAR
  VAR_OUTPUT
    SD1_FaultReset : BOOL := FALSE;
    SD1_O1 : BOOL := FALSE;
    SD1_CI : BOOL := FALSE;
    SD1_CRHO : BOOL := FALSE;
    SD1_II : BOOL := FALSE;
  END_VAR
  VAR
    SD1 : RIN;
  END_VAR
  VAR_OUTPUT
    SD1Clear : BOOL := FALSE;
    AutoOverrideDebounce_DN : BOOL := FALSE;
    AutoOverrideDebounce_ACC : INT := 0;
    AutoOverride_NM : BOOL := FALSE;
    AutoOverride_MMS : BOOL := FALSE;
    ResetReady : BOOL := FALSE;
  END_VAR
  VAR_INPUT
    ResetGrdPB : BOOL;
  END_VAR
  VAR_OUTPUT
    GuardRst_O1 : BOOL := FALSE;
    GuardRst_CI : BOOL := FALSE;
    GuardRst_CRHO : BOOL := FALSE;
    GuardRst_II : BOOL := FALSE;
    GuardReset : BOOL := FALSE;
    ToolMinorEnable : BOOL := FALSE;
    NobotEnable : BOOL := FALSE;
    RobotServoEnable : BOOL := FALSE;
    OneRobotEnable : BOOL := FALSE;
    AutoOverrideDebounce_EN : BOOL := FALSE;
    OverrideLimit_EN : BOOL := FALSE;
    OverrideLimit_ACC : INT := 0;
    OverrideLimit_TT : BOOL := FALSE;
    ToolMajorEnable : BOOL := FALSE;
  END_VAR
  VAR_INPUT
    FlashNorm : BOOL;
  END_VAR
  VAR_OUTPUT
    GuardResetLt : BOOL := FALSE;
  END_VAR
  VAR_IN_OUT
    BackCheck_GateReset : BOOL := FALSE;
    BackCheck_ToolMinorEnable : BOOL := FALSE;
    BackCheck_ToolMajorEnable : BOOL := FALSE;
    BackCheck_NobotEnable : BOOL := FALSE;
    BackCheck_RobotServoEnable : BOOL := FALSE;
  END_VAR
  VAR  (* added by the conversion: wires and edge detectors of the diagram *)
    _MOV_E_Int30_ : ANY;
    _MOV_E_Int30_OUT : INT;
    _MOV_E_Int83_ : ANY;
    _MOV_E_Int83_OUT : INT;
  END_VAR

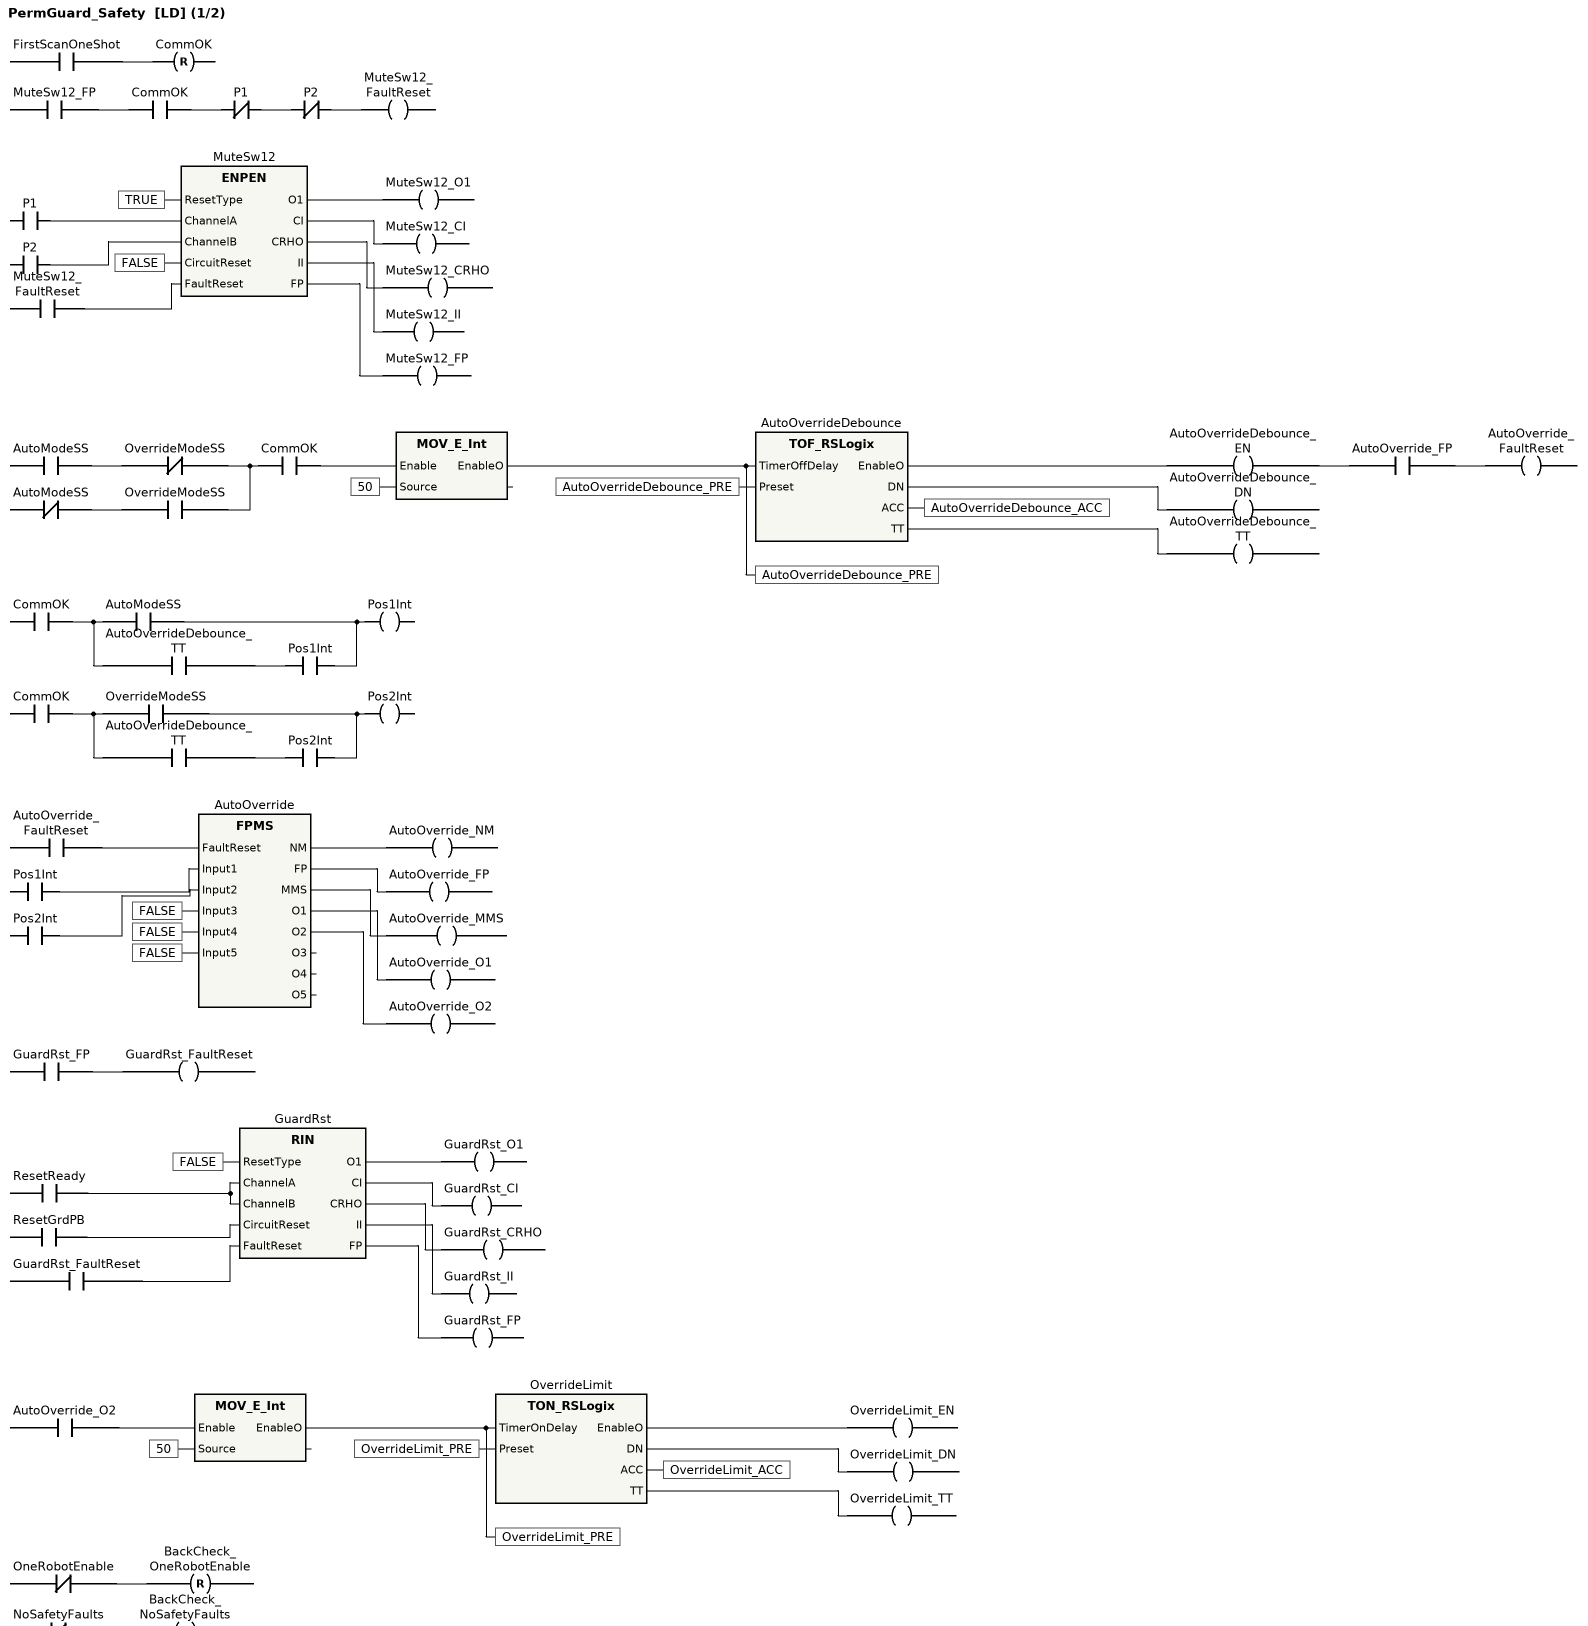
(* LD diagram, written out as Structured Text *)
IF FirstScanOneShot THEN CommOK := FALSE; END_IF;
MuteSw12_FaultReset := MuteSw12_FP AND CommOK AND NOT P1 AND NOT P2;
MuteSw12(ResetType := TRUE, ChannelA := P1, ChannelB := P2, CircuitReset := FALSE, FaultReset := MuteSw12_FaultReset);
MuteSw12_O1 := MuteSw12.O1;
MuteSw12_CI := MuteSw12.CI;
MuteSw12_CRHO := MuteSw12.CRHO;
MuteSw12_II := MuteSw12.II;
MuteSw12_FP := MuteSw12.FP;
MuteSw34_FaultReset := MuteSw34_FP AND CommOK AND NOT P3 AND NOT P4;
MuteSw34(ResetType := TRUE, ChannelA := P3, ChannelB := P4, CircuitReset := FALSE, FaultReset := MuteSw34_FaultReset);
MuteSw34_O1 := MuteSw34.O1;
MuteSw34_CI := MuteSw34.CI;
MuteSw34_CRHO := MuteSw34.CRHO;
MuteSw34_II := MuteSw34.II;
MuteSw34_FP := MuteSw34.FP;
MuteSD := (MuteSw12_O1 OR MuteSw34_O1) AND MutingStatus;
SDMuteLt := MuteSD OR LampTest;
SD1_FaultReset := SD1_FP AND CommOK AND NOT SD1ClearChA AND NOT SD1ClearChB;
SD1(ResetType := TRUE, ChannelA := SD1ClearChA, ChannelB := SD1ClearChB, CircuitReset := FALSE, FaultReset := SD1_FaultReset);
SD1_O1 := SD1.O1;
SD1_CI := SD1.CI;
SD1_CRHO := SD1.CRHO;
SD1_II := SD1.II;
SD1_FP := SD1.FP;
SD1Clear := SD1_O1;
_MOV_E_Int30_OUT := MOV_E_Int(Enable := (AutoModeSS AND NOT OverrideModeSS OR NOT AutoModeSS AND OverrideModeSS) AND CommOK, Source := 50,  => _MOV_E_Int30_);
AutoOverrideDebounce(TimerOffDelay := _MOV_E_Int30_OUT, Preset := AutoOverrideDebounce_PRE);
AutoOverrideDebounce_EN := AutoOverrideDebounce.EnableO;
AutoOverride_FaultReset := AutoOverrideDebounce.EnableO AND AutoOverride_FP;
AutoOverrideDebounce_PRE := _MOV_E_Int30_OUT;
AutoOverrideDebounce_DN := AutoOverrideDebounce.DN;
AutoOverrideDebounce_ACC := AutoOverrideDebounce.ACC;
AutoOverrideDebounce_TT := AutoOverrideDebounce.TT;
Pos1Int := CommOK AND (AutoModeSS OR AutoOverrideDebounce_TT AND Pos1Int);
Pos2Int := CommOK AND (OverrideModeSS OR AutoOverrideDebounce_TT AND Pos2Int);
AutoOverride(FaultReset := AutoOverride_FaultReset, Input1 := Pos1Int, Input2 := Pos2Int, Input3 := FALSE, Input4 := FALSE, Input5 := FALSE);
AutoOverride_NM := AutoOverride.NM;
AutoOverride_FP := AutoOverride.FP;
AutoOverride_MMS := AutoOverride.MMS;
AutoOverride_O1 := AutoOverride.O1;
AutoOverride_O2 := AutoOverride.O2;
ResetReady := (SD1Clear OR MuteSD) AND AutoOverride_O1;
GuardRst_FaultReset := GuardRst_FP;
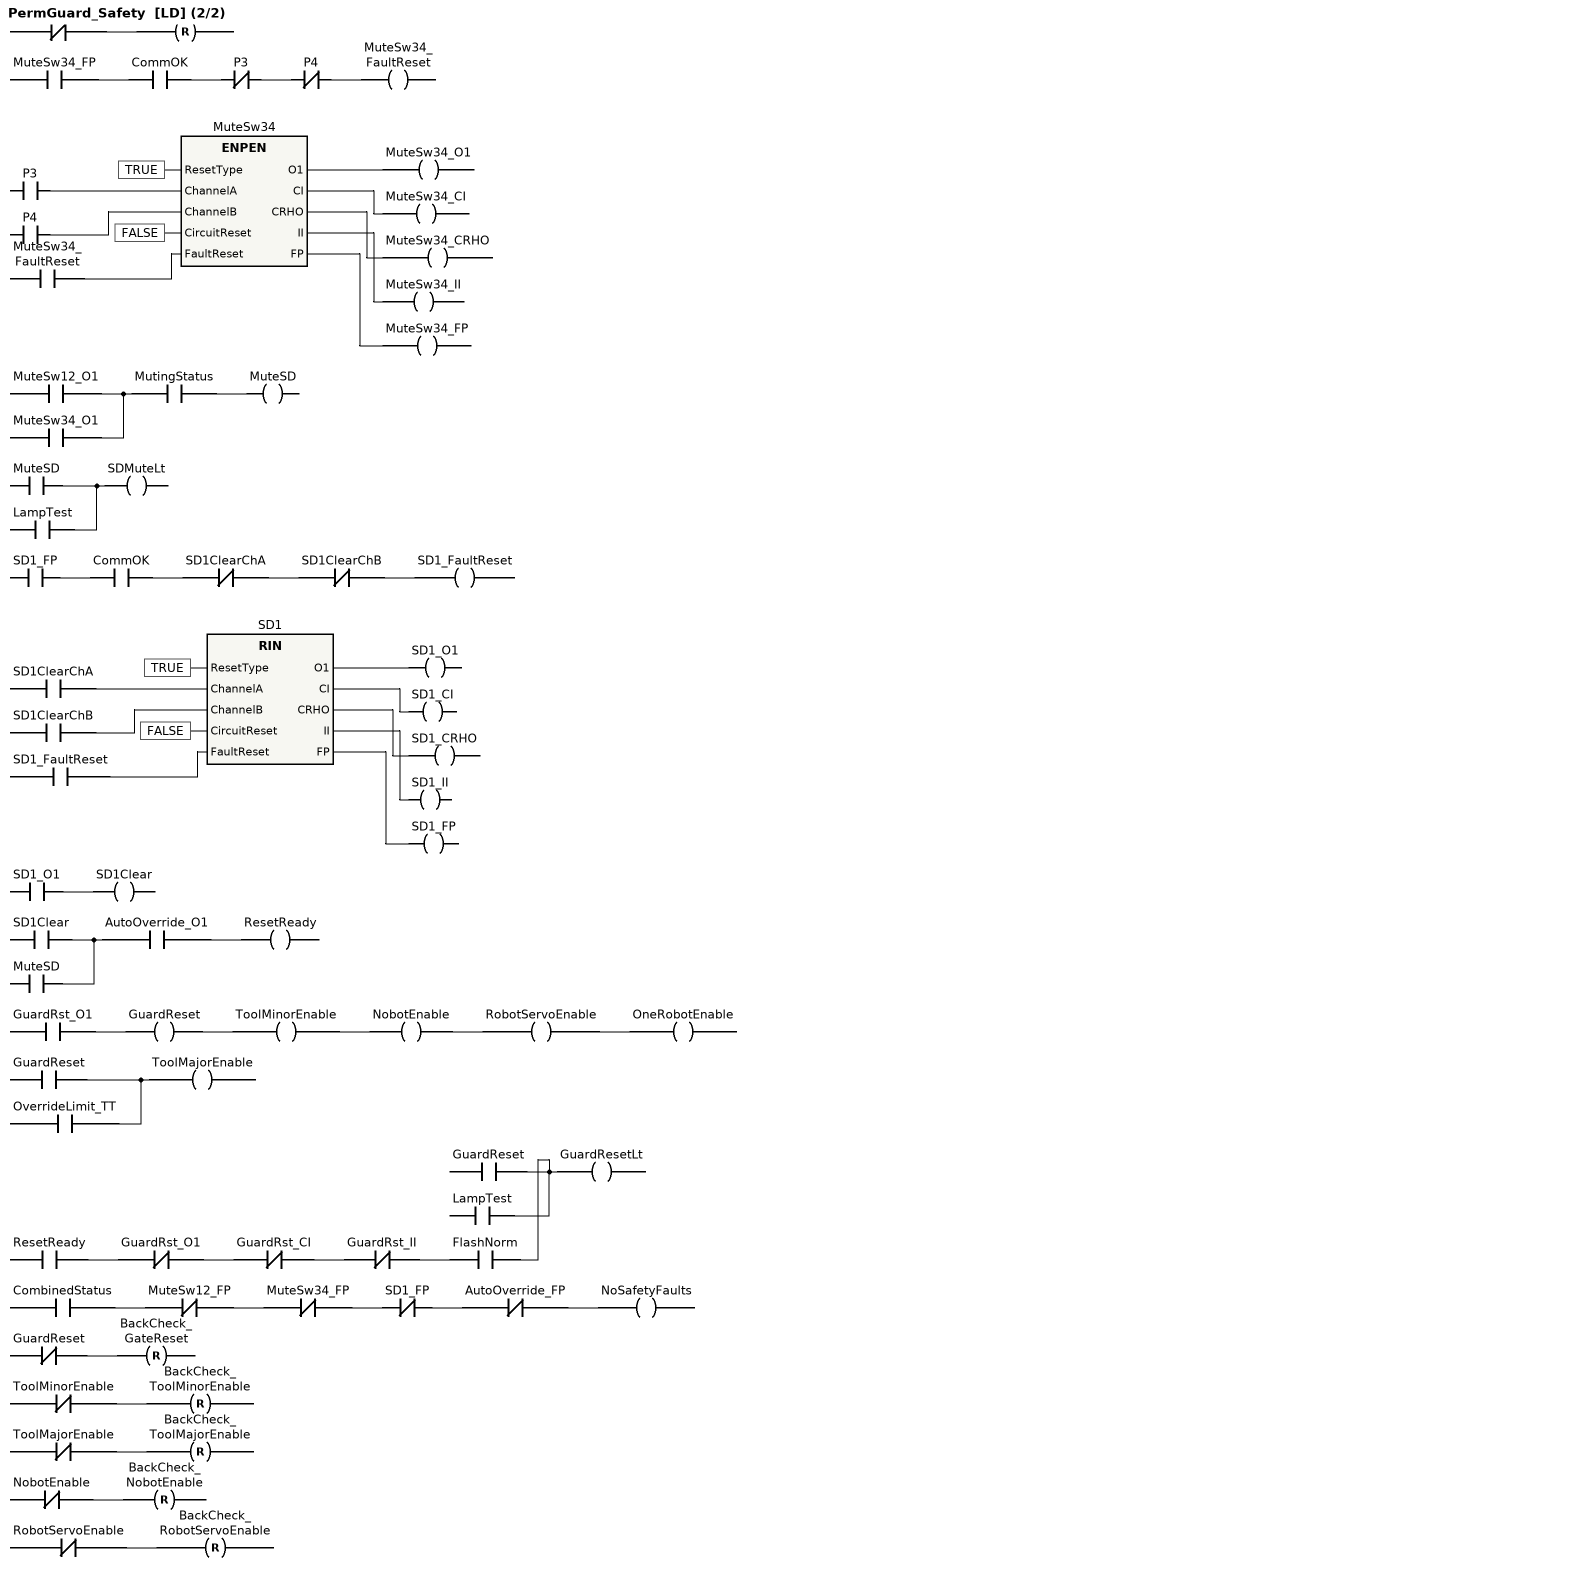
GuardRst(ResetType := FALSE, ChannelA := ResetReady, ChannelB := ResetReady, CircuitReset := ResetGrdPB, FaultReset := GuardRst_FaultReset);
GuardRst_O1 := GuardRst.O1;
GuardRst_CI := GuardRst.CI;
GuardRst_CRHO := GuardRst.CRHO;
GuardRst_II := GuardRst.II;
GuardRst_FP := GuardRst.FP;
GuardReset := GuardRst_O1;
ToolMinorEnable := GuardRst_O1;
NobotEnable := GuardRst_O1;
RobotServoEnable := GuardRst_O1;
OneRobotEnable := GuardRst_O1;
_MOV_E_Int83_OUT := MOV_E_Int(Enable := AutoOverride_O2, Source := 50,  => _MOV_E_Int83_);
OverrideLimit(TimerOnDelay := _MOV_E_Int83_OUT, Preset := OverrideLimit_PRE);
OverrideLimit_EN := OverrideLimit.EnableO;
OverrideLimit_PRE := _MOV_E_Int83_OUT;
OverrideLimit_DN := OverrideLimit.DN;
OverrideLimit_ACC := OverrideLimit.ACC;
OverrideLimit_TT := OverrideLimit.TT;
ToolMajorEnable := GuardReset OR OverrideLimit_TT;
GuardResetLt := GuardReset OR ResetReady AND NOT GuardRst_O1 AND NOT GuardRst_CI AND NOT GuardRst_II AND FlashNorm OR LampTest;
NoSafetyFaults := CombinedStatus AND NOT MuteSw12_FP AND NOT MuteSw34_FP AND NOT SD1_FP AND NOT AutoOverride_FP;
IF NOT GuardReset THEN BackCheck_GateReset := FALSE; END_IF;
IF NOT ToolMinorEnable THEN BackCheck_ToolMinorEnable := FALSE; END_IF;
IF NOT ToolMajorEnable THEN BackCheck_ToolMajorEnable := FALSE; END_IF;
IF NOT NobotEnable THEN BackCheck_NobotEnable := FALSE; END_IF;
IF NOT RobotServoEnable THEN BackCheck_RobotServoEnable := FALSE; END_IF;
IF NOT OneRobotEnable THEN BackCheck_OneRobotEnable := FALSE; END_IF;
IF NOT NoSafetyFaults THEN BackCheck_NoSafetyFaults := FALSE; END_IF;
END_FUNCTION_BLOCK

FUNCTION_BLOCK Emergency_Stop
  VAR_IN_OUT
    EStop_FP : BOOL := FALSE;
  END_VAR
  VAR_INPUT
    CommOK : BOOL;
    NoEStopCHA : BOOL;
    NoEStopCHB : BOOL;
  END_VAR
  VAR_OUTPUT
    EStop_FaultReset : BOOL;
    EStop_O1 : BOOL;
    NoEstop : BOOL;
  END_VAR
  VAR_INPUT
    AutoModeS : BOOL;
    ManModeS : BOOL;
  END_VAR
  VAR_IN_OUT
    AutoMan_FP : BOOL;
  END_VAR
  VAR_OUTPUT
    AutoMan_FaultReset : BOOL;
    AutoManDebounce_PRE : BOOL;
    AutoManDebounce_TT : BOOL;
  END_VAR
  VAR_IN_OUT
    Pos1Int : BOOL;
    Pos2Int : BOOL;
  END_VAR
  VAR_OUTPUT
    AutoMan_O1 : BOOL;
    AutoMan_O2 : BOOL;
    AutoMode : BOOL;
    ManualMode : BOOL;
  END_VAR
  VAR_IN_OUT
    PendantOK_FP : BOOL;
  END_VAR
  VAR_OUTPUT
    PendantOK_FaultReset : BOOL;
  END_VAR
  VAR_INPUT
    E130CREP : BOOL;
    E134CREP : BOOL;
    HMI_Select : BOOL;
  END_VAR
  VAR_IN_OUT
    Selected : BOOL;
  END_VAR
  VAR_INPUT
    HMI_SelectionOK : BOOL;
    Gates_SelectAvail : BOOL;
    EnablePB : BOOL;
  END_VAR
  VAR_IN_OUT
    Enable : BOOL;
    PHMIEnable : BOOL;
    EnableAntiRepeat : BOOL;
  END_VAR
  VAR_OUTPUT
    EnableTmr_PRE : BOOL;
    EnableTmr_EN : BOOL;
    EnableTmr_DN : BOOL;
  END_VAR
  VAR_INPUT
    OneHMIEnabled : BOOL;
    Gates_OneRobotToolMinorReq : BOOL;
    OneHMIMode : BOOL;
  END_VAR
  VAR_OUTPUT
    PendEnable : BOOL;
    PendOk : BOOL;
    RungComment : BOOL;
  END_VAR
  VAR_INPUT
    AlwaysOff : BOOL;
    FltBcn : BOOL;
  END_VAR
  VAR_OUTPUT
    O_FaultLT : BOOL;
  END_VAR
  VAR_INPUT
    ResetLT : BOOL;
  END_VAR
  VAR_OUTPUT
    O_ResetLT : BOOL;
  END_VAR
  VAR_INPUT
    AutoInitLT : BOOL;
  END_VAR
  VAR_OUTPUT
    O_AutoInitLT : BOOL;
  END_VAR
  VAR_INPUT
    CombinedStatus : BOOL;
  END_VAR
  VAR_OUTPUT
    NoSafetyFaults : BOOL;
  END_VAR
  VAR_IN_OUT
    BackCheck_NoEStop : BOOL;
    BackCheck_NoSafetyFaults : BOOL;
  END_VAR

(* LD diagram, written out as Structured Text *)
END_FUNCTION_BLOCK

FUNCTION_BLOCK HMI_Safety_FullAlgorithm
  VAR
    ESTOP_FP : BOOL := FALSE;
  END_VAR
  VAR_IN_OUT
    CommOK : BOOL;
  END_VAR
  VAR_INPUT
    FirstScanOneShot : BOOL;
    NoEStopCHA : BOOL;
    NoEStopCHB : BOOL;
  END_VAR
  VAR
    ESTOP_FaultReset : BOOL;
    ESTOP_O1 : BOOL;
  END_VAR
  VAR_OUTPUT
    NoEstop : BOOL;
  END_VAR
  VAR_INPUT
    AutoModeS : BOOL;
    ManModeS : BOOL;
  END_VAR
  VAR
    AutoMan_FP : BOOL;
    AutoMan_FaultReset : BOOL;
    AutoManDebounce_PRE : BOOL;
    AutoManDebounce_TT : BOOL;
    Pos1Int : BOOL;
    Pos2Int : BOOL;
    AutoMan_O1 : BOOL;
    AutoMan_O2 : BOOL;
  END_VAR
  VAR_OUTPUT
    AutoMode : BOOL;
    ManualMode : BOOL;
  END_VAR
  VAR
    PendantOK_FP : BOOL;
    PendantOK_FaultReset : BOOL;
  END_VAR
  VAR_INPUT
    E130CREP : BOOL;
    E134CREP : BOOL;
    HMI_Select : BOOL;
  END_VAR
  VAR_OUTPUT
    Selected : BOOL;
  END_VAR
  VAR_INPUT
    HMI_SelectionOK : BOOL;
    Gates_SelectAvail : BOOL;
    EnablePB : BOOL;
  END_VAR
  VAR
    Enable : BOOL;
    PHMIEnable : BOOL;
    EnableAntiRepeat : BOOL;
    EnableTmr_PRE : BOOL;
  END_VAR
  VAR_OUTPUT
    EnableTmr_EN : BOOL;
  END_VAR
  VAR
    EnableTmr_DN : BOOL;
  END_VAR
  VAR_INPUT
    OneHMIEnabled : BOOL;
  END_VAR
  VAR
    Gates_OneRobotToolMinorReq : BOOL;
  END_VAR
  VAR_INPUT
    OneHMIMode : BOOL;
  END_VAR
  VAR_OUTPUT
    PendEnable : BOOL;
    PendOk : BOOL;
  END_VAR

(* LD diagram, written out as Structured Text *)
END_FUNCTION_BLOCK

FUNCTION MOV_E_Time : TIME
  VAR_INPUT
    Enable : BOOL;
    Source : TIME;
  END_VAR
  VAR_OUTPUT
    EnableO : BOOL;
  END_VAR

(* LD diagram, written out as Structured Text *)
END_FUNCTION

CONFIGURATION ExampleCell
END_CONFIGURATION
